FUNCTION_BLOCK CL_AxisMaster EXTENDS CL_AxisRobot
var
END_VAR

SUPER^();

METHOD PROTECTED InitDefect : BOOL
sWhichAxis := 'virtual-master';
InitDefect := true;
END_METHOD

END_FUNCTION_BLOCK

(* stored: Version 1.1.0.1, ProductVersion 3.1.4024.12
   POU CL_AxisMaster: Id {f408589f-d93f-4ed2-926a-1d5fc7672154}, SpecialFunc None
   Method InitDefect: Id {66a7c3c9-7aff-4ac1-982c-d54ef8229c1c} *)
